{attribute 'hide'}
{attribute clr [ExcludeFromApiDocumentation()]}
FUNCTION_BLOCK ABSTRACT _internals_TcoSequence EXTENDS TcoSequence

{attribute 'hide'}
METHOD PROTECTED FINAL _Close
THIS^.i_Close();
END_METHOD

{attribute 'hide'}
METHOD PROTECTED FINAL _Open
THIS^.i_Open();
END_METHOD

END_FUNCTION_BLOCK

(* stored: Version 1.1.0.1
   POU _internals_TcoSequence: Id {9ae15687-3f70-0cd0-06b5-b751e2c0a9a9}, SpecialFunc None
   Method _Close: Id {367823d8-9f00-02a0-1a79-3cdd45e38f9e}
   Method _Open: Id {5b3be7a2-ec53-05d4-26ee-6936a7488631} *)
